TYPE ST_Viewer :
STRUCT
	homes	: ARRAY[1..GVL.nHomes] OF ST_Homes;
END_STRUCT
END_TYPE

(* stored: Version 1.1.0.1, ProductVersion 3.1.4024.11
   DUT ST_Viewer: Id {4f320d49-c8fb-4973-aa5c-41ef41d6587c} *)
